TYPE AssemblyComPublishEquipment :
STRUCT

{region "Vertical : Axis"}
  Vertical : ZApplication.AxisComPublish;
  {attribute 'ZId' := '59ce020b-a4f8-4d7a-a0dc-8b778ee4fde8'}
{endregion}

{region "Horizontal : ActuatorDigital"}
  Horizontal : ZApplication.ActuatorDigitalComPublish;
  HorizontalToAssembly : ZApplication.DigitalComPublish;
  HorizontalToTransport : ZApplication.DigitalComPublish;
  HorizontalAtAssembly : ZApplication.DigitalComPublish;
  HorizontalAtTransport : ZApplication.DigitalComPublish;
  {attribute 'ZId' := 'bf04a1fd-9e2a-444c-be25-15a99c5011b8'}
{endregion}

{region "YellowLight : Digital"}
  YellowLight : ZApplication.DigitalComPublish;
  {attribute 'ZId' := 'd8b54b94-4c20-4805-9de3-a35aa5023c5d'}
{endregion}

{region "RedLight : Digital"}
  RedLight : ZApplication.DigitalComPublish;
  {attribute 'ZId' := '810dce14-d302-4e94-b60a-e39841040373'}
{endregion}

{region "GreenLight : Digital"}
  GreenLight : ZApplication.DigitalComPublish;
  {attribute 'ZId' := 'f5a46fca-074f-4557-8a14-cee504d2eb08'}
{endregion}

{region "PneumaticsOk : Digital"}
  PneumaticsOk : ZApplication.DigitalComPublish;
  {attribute 'ZId' := 'e461ecc5-0720-4dc8-ad47-eeb7ce01769f'}
{endregion}

{region "Gripper : ActuatorDigital"}
  Gripper : ZApplication.ActuatorDigitalComPublish;
  GripperAuf : ZApplication.DigitalComPublish;
  {attribute 'ZId' := 'd18888e4-9abb-463d-b01d-e5fd8694a677'}
{endregion}

{attribute '__ZwPlcUnitComDeclaration__'} // Do not remove this attribute! It is used for code generation.

END_STRUCT
END_TYPE

(* stored: Version 1.1.0.1
   DUT AssemblyComPublishEquipment: Id {05a7efca-ddc2-4593-94df-59607caf2f64} *)
